// TIA Portal V17 export
// export: Created 2023-06-23T18:33:39.1307634Z, ExportSetting WithDefaults, DisplayName Totally Integrated Automation Portal, DisplayVersion V17, DisplayName TIA Portal Openness, DisplayVersion V17, DisplayName TIA Portal Version Control Interface, DisplayVersion V17, DisplayName STEP 7 Professional, DisplayVersion V17, DisplayName STEP 7 Safety, DisplayVersion V17, DisplayName WinCC Advanced / Unified PC, DisplayVersion V17
VAR_GLOBAL   // PLC tag table "15_AE1-SA1"
   "iAE1-SA1p" AT %I9.0 : Bool;   // 3
   "iAE1-SA1" AT %I9.1 : Bool;   // 3
   "iAE1-SA1a" AT %I17.2 : Bool;
   "oAE1-SA1p" AT %Q8.3 : Bool;
   "oAE1-SA1" AT %Q8.4 : Bool;
END_VAR
